FUNCTION_BLOCK "FB_AxisPos"
{ S7_Optimized_Access := 'TRUE' }
VERSION : 0.1

// FB_AxisPos: primitiva genérica de posicionamento de UM eixo analógico (interface ESCALAR).
// Comanda o setpoint (o_SetPointCmd -> %QD), lê o feedback (i_PV <- %ID) e gera "em posição"
// (o_InPos) por tolerância + debounce. CONGELA o eixo (segura o último SP) em estado seguro
// ou desabilitado — o freeze é "não reatribuir" o_SetPointCmd (VAR_OUTPUT persiste no DB de
// instância). Instanciada por eixo (X, Z) dentro do FB_PickPlaceSeq (multi-instância);
// NÃO chamar de OB diretamente. Fonte: ARQUITETURA_PickPlace.md §2.7.
    VAR_INPUT
        i_Enable : Bool;    // FALSE = congela (não comanda novo SP)
        i_SafeState : Bool;    // TRUE = congela (estado seguro: não comanda novo destino)
        i_SetPoint : LReal;   // SP desejado (V)
        i_PV : LReal;   // feedback de posição (V)
        i_Tol : LReal;   // tolerância "em posição" (V) — vem de Cfg.PosTol
        i_Debounce : Time;    // estabilização do "em posição" — vem de Cfg.PosDebounce
    END_VAR

    VAR_OUTPUT
        o_SetPointCmd : LReal;   // SP a escrever no %QD (mantém valor em freeze)
        o_InPos : Bool;    // TRUE quando |SPcmd - PV| <= Tol estável por Debounce
    END_VAR

    VAR
        s_tDebounce : TON_TIME;  // debounce do "em posição"
    END_VAR

BEGIN

    REGION Comando de setpoint
    // Comanda novo destino só se habilitado E fora de estado seguro.
    // Caso contrário NÃO reatribui o_SetPointCmd -> ele MANTÉM o último valor (congela).
    // (VAR_OUTPUT de FB persiste no DB de instância entre scans.)
        IF #i_Enable AND NOT #i_SafeState THEN
            #o_SetPointCmd := #i_SetPoint;
        END_IF;
    END_REGION

    REGION Em posicao
    // "em posição" = |SP comandado - PV| <= tolerância, estável por Debounce.
    // Usa o_SetPointCmd (o destino atual, mesmo congelado), não i_SetPoint.
        #s_tDebounce(IN := ABS(#o_SetPointCmd - #i_PV) <= #i_Tol,
        PT := #i_Debounce);
        #o_InPos := #s_tDebounce.Q;
    END_REGION

END_FUNCTION_BLOCK